Fanuc KAREL source: kt00888.KL

-- PROVISIONAL review KL for V770-1; original PC SHA256 3cca1a3e74affed25e9abc5ff40b397615435ce5a97bab7f22854b77415bd747
-- Incomplete behavior may be omitted. Consult companion uncertainty JSON. Do not deploy.
PROGRAM KT00888
%NOLOCKGROUP
-- UNRESOLVED_DECL P1 type=000101
-- UNRESOLVED_DECL P2 type=000101
-- UNRESOLVED_DECL OUT type=000101
BEGIN
  -- UNRESOLVED_PC offsets 5-32; opcodes 27,22,1C,76,7E,4A
  -- UNRESOLVED_PC offsets 37-41; opcodes 7F
END KT00888
